{attribute 'GeneratedUsingTerminal: EL7211-0010-0032'}
{attribute addProperty BoxType "EL7211-0010-0032"}
{attribute addProperty Id "Following_error_actual_valueAT %I*DINT4"}
{attribute addProperty CRC "1520640191"}
{attribute addProperty Size "4"}
TYPE DRV_Following_error_actual_value_5AA320BF EXTENDS TcoIo.InputBase_8311D824 :
STRUCT
	{attribute addProperty Name "Following_error_actual_value"}
	Following_error_actual_value AT %I* : DINT;
END_STRUCT
END_TYPE

(* stored: Version 1.2.0.0, ProductVersion 3.1.4024.11
   DUT DRV_Following_error_actual_value_5AA320BF: Id {aa5ae66d-bcd7-0f09-3049-d09a87b8ab9d} *)
